FUNCTION_BLOCK T_TestEvent EXTENDS T_EventBase 
VAR
    Handler : I_TestEventHandler;
END_VAR

METHOD PRIVATE CallHandler
VAR_INPUT
    HandlerBase : I_EventHandlerBase;
    EventArgs   : I_StreamReader;
END_VAR
IF __QUERYINTERFACE(HandlerBase,Handler) THEN
    Handler.OnCustomEvent(EventArgs);
//ELSE
//    tcl_BaseClasses.F_LogError('Event Handling',F_FormatStringEx1('Error raising %s - invalid handler',EventName));
END_IF
END_METHOD

METHOD IsHandlerSupported : BOOL
VAR_INPUT
    HandlerBase : I_EventHandlerBase;
END_VAR
IF __QUERYINTERFACE(HandlerBase,Handler) THEN
    IsHandlerSupported := TRUE;
END_IF
END_METHOD

END_FUNCTION_BLOCK

(* stored: Version 1.1.0.1, ProductVersion 3.1.4024.4
   POU T_TestEvent: Id {71c3a7a7-a6cb-4c04-8081-db6bdc9f902a}, SpecialFunc None
   Method CallHandler: Id {cd89012e-08a5-4a72-84fb-010eeebb5ae8}
   Method IsHandlerSupported: Id {32a98609-17c8-410a-8426-dbca206a6c1b} *)
